FUNCTION_BLOCK SP_MoveNeedleDown (* MoveNeedleDown parameters (Distance [mm] 0.0..50.0, default 50.0): OPC UA IDs, range check and latching *)
  (* Standard: 61499-2 *)
  (* Version 0.1, 2026-09-28, Project contributors, AAU Smart Production Lab *)
  PACKAGE filler;
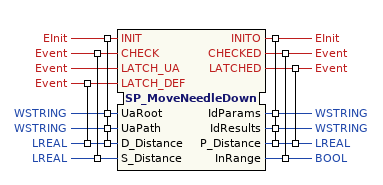
  EVENT_INPUT
    INIT : EInit WITH UaRoot, UaPath, D_Distance;
    CHECK WITH S_Distance;
    LATCH_UA;
    LATCH_DEF WITH D_Distance;
  END_EVENT
  EVENT_OUTPUT
    INITO : EInit WITH IdParams, IdResults, P_Distance;
    CHECKED WITH InRange;
    LATCHED WITH P_Distance;
  END_EVENT
  VAR_INPUT
    UaRoot : WSTRING;
    UaPath : WSTRING;
    D_Distance : LREAL;
    S_Distance : LREAL;
  END_VAR
  VAR_OUTPUT
    IdParams : WSTRING;
    IdResults : WSTRING;
    P_Distance : LREAL;
    InRange : BOOL;
  END_VAR
  EC_STATES
    INIT : INIT -> INITO;
    CHECK : CHECK -> CHECKED;
    LATCH_UA : LATCH_UA -> LATCHED;
    LATCH_DEF : LATCH_DEF -> LATCHED;
  END_STATES
  ALGORITHM INIT IN ST:
IdParams := CONCAT(CONCAT(CONCAT("opc_ua[WRITE;", CONCAT(UaRoot, UaPath)), "/Parameters/Distance"), "]");
IdResults := "";
P_Distance := D_Distance;
  END_ALGORITHM
  ALGORITHM CHECK IN ST:
InRange := (S_Distance >= 0.0) AND (S_Distance <= 50.0);
  END_ALGORITHM
  ALGORITHM LATCH_UA IN ST:
P_Distance := S_Distance;
  END_ALGORITHM
  ALGORITHM LATCH_DEF IN ST:
P_Distance := D_Distance;
  END_ALGORITHM
END_FUNCTION_BLOCK
